(* IEC 61131-3 sources: AcpTrakStarwheel/Starlib, 9 files *)

(* ---- Types.typ ---- *)
TYPE
	FindClosestPcketSynReturnType : 	STRUCT
		ClosestPocket : UINT;
		NextClosestPocket : UINT;
	END_STRUCT;
END_TYPE

(*Star Target Calculations*)

TYPE
	slStarCalcTargetParType : 	STRUCT  (*Pocket sync position calculation parameters*)
		StarwheelRadius : REAL; (*Radius of the starwheel in mm*)
		StarwheelPeriod : REAL; (*Period of the starwheel in degrees*)
		StarwheelPocketCount : USINT; (*Number of pockets on the starwheel*)
		SectorTangentPos : REAL; (*Tangent position of the starwheel on the Trak sector*)
		DeltaT : TIME; (*Delay time to compensate in ms*)
	END_STRUCT;
	slStarCalcTargetInternalType : 	STRUCT  (*Internal Data*)
		TargetIndex : USINT; (*Index to generate a position for*)
		PeriodCount : INT; (*Number of periods being monitored*)
		CurrentStarwheelPeriod : INT; (*The current period of the target*)
		MultiturnPosition : REAL; (*The current multiturn position of the starwheel*)
		StarPosPredict : REAL; (*Starwheel predicted position*)
		OldStarPosPredict : REAL; (*Previously recorded predicted starwheel position*)
		AngleOffset : REAL; (*Angle offset of the starwheel compensating for pocket and period*)
		PocketAngle : REAL; (*Angle of the monitored pocket*)
		TrakSyncPosRaw : REAL; (*Raw trak position not accounting for the tangent position*)
		PerformCalculation : BOOL; (*Perform calculation while true*)
		State : slStarCalcTargetStateEnum; (*State of execution*)
	END_STRUCT;
	slStarCalcTargetStateEnum :
		( (*State of execution*)
		slTARGET_CALC_STATE_IDLE, (*Idle state*)
		slTARGET_CALC_STATE_RUN, (*Run state*)
		slTARGET_CALC_STATE_ERROR (*Error state*)
		);
END_TYPE

(*Star Pocket Sync*)

TYPE
	slStarPocketSyncParType : 	STRUCT  (*Pocket Sync Parameters*)
		StarCalcTarget : slStarCalcTargetParType; (*Calculation parameters*)
		CycPos : slStarPocketCycPosParType; (*Cyclic position parameters*)
		ResizeStart : McAcpTrakShResizeParamType; (*Resize dimensions at start of synchronization*)
		ResizeEnd : McAcpTrakShResizeParamType; (*Resize dimensions at end of synchronization*)
		Release : slStarPocketSyncReleaseParType; (*Release Parameters*)
	END_STRUCT;
	slStarPocketCycPosParType : 	STRUCT  (*Cyclic Position parameters*)
		AdvancedParameters : McAdvMoveCycParType; (*Advanced parameters*)
		InterpolationMode : McIplModeEnum; (*Interpolation mode*)
	END_STRUCT;
	slStarPocketSyncReleaseParType : 	STRUCT  (*Release motion parameters*)
		Position : LREAL; (*Release position on trak*)
		ResizePosition : LREAL; (*Resize position on trak after release*)
		Velocity : REAL; (*Release Velocity*)
		Acceleration : REAL; (*Release Acceleration*)
		Deceleration : REAL; (*Release Deceleration*)
		Jerk : REAL; (*Release Jerk*)
		Direction : McDirectionEnum; (*Release Direction*)
		BufferMode : McBufferModeEnum; (*Release Buffer Mode*)
	END_STRUCT;
	slStarPocketSyncInternalType : 	STRUCT  (*Internal Data*)
		StarCalcTarget : slStarCalcTarget; (*Calculate the sync position*)
		CycPos : MC_BR_ElasticMoveCycPos_AcpTrak; (*Synchronize the shuttle ot the position*)
		ShReadInfo : MC_BR_ShReadInfo_AcpTrak; (*Read shuttle information for its position*)
		MoveVel : MC_BR_ElasticMoveVel_AcpTrak; (*Release the shuttle from synchronization*)
		Resize : MC_BR_ShResize_AcpTrak; (*Resize the shuttle at start*)
		State : slStarPocketSyncStateEnum; (*State of execution*)
	END_STRUCT;
	slStarPocketSyncStateEnum :
		( (*State of execution*)
		slPOCKET_SYN_STATE_IDLE, (*Idle state*)
		slPOCKET_SYN_STATE_WAIT_SYNC, (*Wait for sync*)
		slPOCKET_SYN_STATE_RESIZE_START, (*Resize shuttle for start of sync*)
		slPOCKET_SYN_STATE_SYNC, (*Perform synchronization*)
		slPOCKET_SYN_STATE_RELEASE, (*Release shuttle*)
		slPOCKET_SYN_STATE_WAIT_RESIZE, (*Wait for the shuttle to reach the position to resize*)
		slPOCKET_SYN_STATE_RESIZE_END, (*Resize shuttle for end of sync*)
		slPOCKET_SYN_STATE_DONE, (*Star wheel operation complete*)
		slPOCKET_SYN_STATE_RESET_FB, (*Reset function blocks*)
		slPOCKET_SYN_STATE_WAIT_NOT_BUSY, (*Wait for function blocks to report not busy*)
		slPOCKET_SYN_STATE_ERROR (*Error state*)
		);
END_TYPE

(*Star Recovery*)

TYPE
	slStarRecoveryParType : 	STRUCT  (*Star recovery parameters*)
		ResizeStart : McAcpTrakShResizeParamType; (*Resize dimensions at start of synchronization*)
		ResizeEnd : McAcpTrakShResizeParamType; (*Resize dimensions at end of synchronization*)
		SyncFurtherInEnabled : BOOL;
		Release : slStarRecoveryParReleaseType; (*Recovery Release Parameters*)
		ProcessPointStartPosition : LREAL; (*Position on the sector of the process point that starts the synchronization*)
		StartOffset : LREAL; (*Offset from the process point before synchronizing*)
		PocketErrorTolerance : LREAL; (*Allowed pocket error tolerance*)
		UserData : slStarRecoveryParUserDataType; (*UserData parameters*)
		Backup : slStarRecoveryParBackupType;
		ShExtentToFront : LREAL;
		SectorTangentPos : REAL;
		MeshZoneStartPos : LREAL; (*Starwheel dimensions*)
		MeshZoneEndPos : LREAL;
	END_STRUCT;
	slStarRecoveryParBackupType : 	STRUCT  (*Recovery Release Parameters*)
		BackupTolerance : LREAL;
		ProcessPointStart : McProcessPointType; (*Position on the sector of the process point that starts the synchronization*)
		MoveToBarAcceleration : REAL;
		MoveToBarDeceleration : REAL;
		MoveToBarVelocity : REAL;
	END_STRUCT;
	slStarRecoveryParUserDataType : 	STRUCT  (*UserData parameters*)
		UserDataAddress : UDINT; (*Pointer to the user data buffer*)
		UserDataSize : UDINT; (*Size of the user data buffer*)
		SrcUserDataWriteAddress : UDINT; (*Source of the data to write to the user data buffer*)
		DstUserDataWriteAddress : UDINT; (*Destination within the user data buffer to write*)
		UserDataWriteSize : UDINT; (*Size of the data to write to the user data buffer*)
	END_STRUCT;
	slStarRecoveryParReleaseType : 	STRUCT  (*Recovery Release Parameters*)
		Position : LREAL; (*Release position of the starwheel*)
		Velocity : REAL; (*Recovery Velocity*)
		Acceleration : REAL; (*Recovery Acceleration*)
		Deceleration : REAL; (*Recovery Deceleration*)
		DestinationSector : McSectorType; (*Recovery Destination Sector*)
	END_STRUCT;
	slStarRecoveryInternalType : 	STRUCT  (*Internal Data*)
		Handle : UDINT; (*Handle to the starwheel internal data*)
		SecGetShuttle : MC_BR_SecGetShuttle_AcpTrak; (*Get shuttles on the sector*)
		ShResize : MC_BR_ShResize_AcpTrak; (*Resize shuttle*)
		RoutedMoveVel : MC_BR_RoutedMoveVel_AcpTrak; (*Send shuttle*)
		RoutedMoveAbs : MC_BR_RoutedMoveAbs_AcpTrak;
		ElasticMoveVel : MC_BR_ElasticMoveVel_AcpTrak; (*Send the shuttle*)
		ElasticMoveAbs : MC_BR_ElasticMoveAbs_AcpTrak;
		ShCopyUserData : MC_BR_ShCopyUserData_AcpTrak; (*Copy user data*)
		AsmGetInfo : MC_BR_AsmGetInfo_AcpTrak; (*Used to see if sectors are being simulated*)
		BarrierCmd : MC_BR_BarrierCommand_AcpTrak;
		OldRemainingCount : UINT; (*Previously recorded remaining count*)
		Data : slStarRecoveryInternalDataType; (*Data*)
		State : slStarRecoveryStateEnum; (*State of execution*)
		i : USINT; (*Index*)
	END_STRUCT;
	slStarRecoveryInternalDataFIType : 	STRUCT
		CurrentPocketIndex : UINT; (*Current pocket index being evaluated*)
	END_STRUCT;
	slStarRecoveryInternalDataType : 	STRUCT  (*Recovery data*)
		Init : slStarRecoverylDataInitType; (*Initial recovery data*)
		Mesh : slStarRecoveryDataMeshType;
		Sync : slStarRecoveryDataSyncType; (*Sync recovery data*)
		Backup : slStarRecoveryDataBackupType; (*Backup recovery data*)
		UserData : slStarRecoveryDataUserDataType;
		SyncFurtherIn : slStarRecoveryInternalDataFIType;
		PocketWidth : LREAL; (*Width of a pocket on the starwheel*)
	END_STRUCT;
	slStarRecoveryDataSyncFurInType : 	STRUCT
		LastSyncedPocket : USINT; (*Next open pocket available to sync further in*)
		LastSyncedPocketValid : BOOL;
	END_STRUCT;
	slStarRecoveryDataUserDataType : 	STRUCT
		UserDataWriteCount : UINT;
	END_STRUCT;
	slStarRecoverylDataInitType : 	STRUCT  (*Intial recovery data*)
		ShuttlePos : ARRAY[0..slMAX_SH_IDX_IN_SEC]OF LREAL; (*Shuttle positions found at initialization*)
		ShuttleAxis : ARRAY[0..slMAX_SH_IDX_IN_SEC]OF McAxisType; (*Shuttle axes found at initialization*)
		NumShuttles : UINT; (*Number of shuttles found at initialization*)
		ShuttleEvalCount : USINT; (*Number of shuttles found at initialization that have been evalueated*)
	END_STRUCT;
	slStarRecoveryDataMeshType : 	STRUCT  (*Sync recovery data*)
		PocketEvalIndex : UINT; (*Pocket index to evaluate*)
		PocketEvalIndexValid : BOOL;
		NextClosestPocketIndex : UINT;
		ClosestPocketTaken : BOOL;
		NextClosestPocketTaken : BOOL;
		PocketEvalCount : USINT; (*Number of pockets evaluated*)
		Axes : ARRAY[0..slMAX_SH_IDX_IN_SEC]OF McAxisType; (*Sync axes*)
		ShuttleErrors : ARRAY[0..slMAX_SH_IDX_IN_SEC]OF LREAL;
		PocketIndices : ARRAY[0..slMAX_SH_IDX_IN_SEC]OF UINT; (*Pocket indices assigned to the sync axes*)
		ShuttleError : LREAL; (*Distance from shuttle to pocket*)
		ShuttleErrorNew : LREAL; (*New distance from shuttle to pocket*)
		NextClosestPocketError : LREAL;
		RecoveredCount : UINT; (*Number of shuttles recovered*)
	END_STRUCT;
	slStarRecoveryDataSyncType : 	STRUCT  (*Sync recovery data*)
		PocketEvalIndex : UINT; (*Pocket index to evaluate*)
		PocketEvalIndexValid : BOOL;
		NextClosestPocketIndex : UINT;
		ClosestPocketTaken : BOOL;
		NextClosestPocketTaken : BOOL;
		PocketEvalCount : USINT; (*Number of pockets evaluated*)
		Axes : ARRAY[0..slMAX_SH_IDX_IN_SEC]OF McAxisType; (*Sync axes*)
		ShuttleErrors : ARRAY[0..slMAX_SH_IDX_IN_SEC]OF LREAL;
		PocketIndices : ARRAY[0..slMAX_SH_IDX_IN_SEC]OF UINT; (*Pocket indices assigned to the sync axes*)
		ShuttleError : LREAL; (*Distance from shuttle to pocket*)
		ShuttleErrorNew : LREAL; (*New distance from shuttle to pocket*)
		RecoveredCount : UINT; (*Number of shuttles recovered*)
		ShuttlePos : ARRAY[0..slMAX_SH_IDX_IN_SEC]OF LREAL; (*Shuttle positions found at initialization*)
		SyncFurtherIn : slStarRecoveryDataSyncFIType;
		NextClosestPocketError : LREAL;
	END_STRUCT;
	slStarRecoveryDataSyncFIType : 	STRUCT
		ClosestPocketToMeshFound : BOOL;
		ClosestPocketToMesh : UINT;
		NoClosestPocketFound : BOOL;
		FirstPocketInMeshIndex : UINT;
		FirstShuttleInMeshError : LREAL;
		FirstSyncPocketError : LREAL;
	END_STRUCT;
	slStarRecoveryDataBackupType : 	STRUCT  (*Backup recovery data*)
		EvalCount : USINT; (*Number of shuttles evaluated*)
		Axes : ARRAY[0..slMAX_SH_IDX_IN_SEC]OF McAxisType; (*Axes found in the backup area*)
		Positions : ARRAY[0..slMAX_SH_IDX_IN_SEC]OF LREAL;
		RecoveredCount : USINT; (*Number of shuttles recovered*)
		IsBeforeBarrier : ARRAY[0..slMAX_SH_IDX_IN_SEC]OF BOOL; (*Indicates if a shuttle is in the backup zone but before the barrier (have to move to gaurantee it won't get stuck at the barrier)*)
		MovedToBarrier : ARRAY[0..slMAX_SH_IDX_IN_SEC]OF BOOL; (*Indicated if a shuttle has been moved to the barrier location*)
		SyncFurtherIn : slStarRecoveryDataBackupFIType;
		Position : LREAL;
		PocketOvertakeIndex : UINT;
	END_STRUCT;
	slStarRecoveryDataBackupFIType : 	STRUCT  (*Sync further in type for backup zone*)
		CurrentPocketIndex : UINT; (*Current pocket index being evaluated*)
		SyncFurtherInFinished : BOOL; (*All shuttles in backup zone have synced to the closest pockets possible*)
	END_STRUCT;
	slStarRecoveryStateEnum :
		( (*State of execution*)
		slREC_STATE_IDLE, (*Idle state*)
		slREC_STATE_CHECK_SECTOR_SIM,
		slREC_STATE_GET_SHUTTLES, (*Get shuttles on the sector*)
		slREC_STATE_ATTACH_TO_SECTOR,
		slREC_STATE_GET_SHUTTLES_NEXT, (*Get the next shuttle on the sector*)
		slREC_STATE_RELEASE_ZONE_CHECK, (*Check for shuttles in the release zone*)
		slREC_STATE_RELEASE_ZONE_RESIZE, (*Resize shuttles in the release zone*)
		slREC_STATE_RELEASE_ZONE_SEND, (*Send shuttles in the release zone*)
		slREC_STATE_RELEASE_ZONE_NEXT, (*Get the next shuttle in the release zone*)
		slREC_STATE_MESH_ZONE_CHECK, (*Check for shuttles in the sync zone*)
		slREC_STATE_MESH_ZONE_TARGET, (*Assign target for sync*)
		slREC_STATE_MESH_ZONE_RESIZE, (*Resize shuttles*)
		slREC_STATE_MESH_ZONE_NEXT, (*Get the next shuttle in the sync zone*)
		slREC_STATE_SYN_ZONE_CHECK, (*Check for shuttles in the sync zone*)
		slREC_STATE_SYN_ZONE_TARGET, (*Assign target for sync*)
		slREC_STATE_SYN_ZONE_RESIZE, (*Resize shuttles*)
		slREC_STATE_SYN_ZONE_NEXT, (*Get the next shuttle in the sync zone*)
		slREC_STATE_BACKUP_ZONE_CHECK, (*Check for shuttles in the backup zone*)
		slREC_STATE_PBACKUP_ZONE_RSIZE, (*Resize shuttles in the backup zone*)
		slREC_STATE_PBACKUP_ZONE_SEND, (*Send shuttles in the backup zone*)
		slREC_STATE_PBACKUP_ZONE_NEXT, (*Get the next shuttle in the backup zone*)
		slREC_STATE_PBCKUP_ZNE_USR_DATAG, (*Get the next shuttle in the backup zone*)
		slREC_STATE_SYN_ZONE_SYNC, (*Sync shuttles in the sync zone*)
		slREC_STATE_MESH_ZONE_SYNC, (*Sync shuttles in the sync zone*)
		slREC_STATE_SYN_GET_USERDATA, (*Get sync zone userdata*)
		slREC_STATE_SYN_SET_USERDATA, (*Set sync zone userdata*)
		slREC_STATE_BACKUP_ZONE_TARGET, (*Wait for a target for shuttle in backup zone*)
		slREC_STATE_BACKUP_ZONE_BAROPEN, (*Wait for a target for shuttle in backup zone*)
		slREC_STATE_BACKUP_ZONE_MOVBAR,
		slREC_STATE_BACKUP_ZONE_BARCLOSE,
		slREC_STATE_BACKUP_ZONE_SYNC, (*Sync shuttle in backup zone to target*)
		slREC_STATE_BACKUP_ZONE_SYNC_FI, (*Backup zone sync further in*)
		slREC_STATE_BACKUP_GET_USERDATA, (*Get backup zone userdata*)
		slREC_STATE_BACKUP_SET_USERDATA, (*Set backup zone userdata*)
		slREC_STATE_GET_USERDATA,
		slREC_STATE_SET_USERDATA,
		slREC_STATE_FI_WAIT_SHUTTLE, (*Wait for a new shuttle to come by*)
		slREC_STATE_DONE, (*Recovery is complete*)
		slREC_STATE_WAIT_NOT_BUSY, (*Wait for function blocks to report not busy*)
		slREC_STATE_ERROR (*Error state*)
		);
END_TYPE

(*Star Sync*)

TYPE
	slStarSyncParType : 	STRUCT  (*Pocket Queue Parameters*)
		Landing : slStarSyncLandingParType; (*Landing parameters*)
		Starting : slStarSyncStartingParType; (*Starting parameters*)
		Staging : slStarSyncStagingParType; (*Staging parameters*)
		StartOffset : LREAL; (*Offset from the staging position before synchronizing*)
		SyncPar : slStarPocketSyncParType; (*Synchronization parameters*)
		Recovery : slStarSyncRecoveryParType; (*Star parameters for recovery*)
		Skip : slStarSyncSkipParType; (*Skip parameters*)
		ShExtentToFront : LREAL;
	END_STRUCT;
	slStarSyncLandingParType : 	STRUCT  (*Landing parameters*)
		Position : LREAL; (*Target Position*)
		Velocity : REAL; (*Target Velocity*)
		Acceleration : REAL; (*Target Acceleration*)
		Deceleration : REAL; (*Target Deceleration*)
		AdvancedParameters : McAcpTrakAdvRouteParType; (*Advanced move parameters*)
	END_STRUCT;
	slStarSyncStartingParType : 	STRUCT  (*Starting parameters*)
		Position : LREAL; (*Target Position*)
		Velocity : REAL; (*Target Velocity*)
	END_STRUCT;
	slStarSyncStagingParType : 	STRUCT  (*Staging parameters*)
		Position : LREAL; (*Target Position*)
		Velocity : REAL; (*Target Velocity*)
		Acceleration : REAL; (*Target Acceleration*)
		Deceleration : REAL; (*Target Deceleration*)
	END_STRUCT;
	slStarSyncRecoveryParType : 	STRUCT  (*Star parameters for recovery*)
		Release : slStarSyncRecoveryReleaseType; (*Release parameters*)
		UserData : slStarRecoveryParUserDataType; (*User data buffer data for successful recovery*)
		SyncFurtherInEnabled : BOOL;
		PocketErrorTolerance : LREAL; (*Pocket error tolerance for resynchronization*)
		MoveToBarVelocity : REAL;
		MoveToBarAcceleration : REAL;
		MoveToBarDeceleration : REAL;
		BackupTolerance : LREAL;
	END_STRUCT;
	slStarSyncRecoveryReleaseType : 	STRUCT  (*Release parameters*)
		Velocity : REAL; (*Recovery Velocity*)
		Acceleration : REAL; (*Recovery Acceleration*)
		Deceleration : REAL; (*Recovery Deceleration*)
		DestinationSector : McSectorType; (*Recovery Destination Sector*)
	END_STRUCT;
	slStarSyncSkipParType : 	STRUCT  (*Skip parameters*)
		NumSkips : USINT; (*Number of skips if skipping is enabled*)
		NumDisabled : USINT; (*Number of disabled pockets*)
		DisabledIdx : ARRAY[0..slMAX_DISABLE_POCKET_IDX]OF USINT; (*Disabled pockets*)
	END_STRUCT;
	slStarSyncCalcDataType : 	STRUCT
		StarPosPredict : REAL; (*Current starwheel position + predictive compensation*)
		CurrentStarwheelPeriod : INT; (*Current period of the 'real' starwheel, used to calculate a multiturn position*)
		MultiturnPosition : REAL; (*Current position of the 'virtual' starwheel*)
	END_STRUCT;
	slStarSyncInternalType : 	STRUCT  (*Internal Data*)
		TypeID : UDINT; (*Internal data type ID*)
		ErrorID : DINT; (*Last recorded error ID*)
		Recovery : slStarRecovery; (*Recovery process*)
		RecoveryPar : slStarRecoveryParType; (*Recovery parameters*)
		MaxTargetIndex : USINT; (*Highest pocket sync target index used*)
		LandingBuffer : tbAsyncShuttleBufferType; (*Buffer of shuttles that are landing on the sector*)
		StagingBuffer : tbAsyncShuttleBufferType; (*Buffer of shuttles that are being staged*)
		LandingBufferMan : tbRoutedMoveVelTrgBuffer; (*Landing shuttle buffer manager*)
		LandingBufferPar : tbRtdMvVelTrgBufferParType; (*Landing buffer parameters*)
		StagingBufferMan : tbElasticMoveAbsPosBuffer; (*Staging shuttle buffer manager*)
		StagingBufferPar : tbElaMvAbsPosBufferParType; (*Staging buffer parameters*)
		PocketSync : ARRAY[0..slMAX_TARGET_IDX]OF slStarPocketSync; (*Pocket Sync Targets*)
		LastPocketActiveState : ARRAY[0..slMAX_TARGET_IDX]OF BOOL; (*Capture the last pocket sync active state*)
		LastTargetPosition : ARRAY[0..slMAX_TARGET_IDX]OF REAL; (*Last observed target position for each target*)
		NextSyncTarget : UINT; (*Next target to sync shuttle with*)
		NewDisabledOvertake : BOOL; (*A disabled target position has passed the synchronization threshold*)
		NewOvertakeDetected : BOOL; (*A target position has passed the synchronization threshold*)
		State : slStarSyncStateEnum; (*State of execution*)
		SkipCount : USINT; (*Number of pockets skipped*)
		PocketDisabled : BOOL; (*Current target pocket is disabled*)
		PeriodCount : USINT; (*Number of periods to monitor*)
		i : UINT; (*Index*)
		n : USINT; (*Index*)
		PocketSyncBusy : BOOL; (*Temporary variable to determine if a pocket sync is still busy*)
		PocketSyncError : BOOL; (*Temporary variable to determine if a pocket sync has an error*)
		PocketSyncErrorID : DINT; (*Temporary variable to determine the pocket sync error ID*)
		NextSyncFITarget : UINT; (*Next sync further in target found*)
		SyncFurtherInDone : BOOL;
		MeshZoneStartPos : LREAL;
		MeshZoneEndPos : LREAL;
		PocketWidth : LREAL;
		RecoveryDone : BOOL;
		StarCalcData : slStarSyncCalcDataType; (*Includes Calc Target information that is Starwheel-specific, rather than Pocket-specific*)
		OldStarPosPredict : REAL; (*Star Position, including predictive compensation, from last cycle*)
		Status : DINT; (*Status*)
	END_STRUCT;
	slStarSyncStateEnum :
		( (*State of execution*)
		slSTAR_STATE_INIT, (*Initialize handle and data*)
		slSTAR_STATE_IDLE, (*Idle state*)
		slSTAR_STATE_RECOVER, (*Recover shuttles*)
		slSTAR_STATE_WAIT_TARGET, (*Wait for the next target to arrive*)
		slSTAR_STATE_WAIT_SHUTTLE, (*Wait for the next shuttle to arrive*)
		slSTAR_STATE_SYNC, (*Sync shuttle to pocket*)
		slSTAR_STATE_RESET_FB, (*Reset function blocks*)
		slSTAR_STATE_WAIT_NOT_BUSY, (*Wait for function blocks to report not busy*)
		slSTAR_STATE_ERROR (*An error occurred*)
		);
END_TYPE

(*Get Shuttle*)

TYPE
	slStarGetShuttleInternalType : 	STRUCT  (*Internal Data*)
		i : USINT; (*Index*)
		Present : BOOL; (*Temporary shuttle presence*)
		Axis : McAxisType; (*Temporary Axis Handle*)
		Position : REAL; (*Temporary Position*)
	END_STRUCT;
END_TYPE

(*Star Sync Diagnostics*)

TYPE
	slStarDiagType : 	STRUCT  (*Output starwheel diagnostics*)
		AngleOffset : ARRAY[0..slMAX_TARGET_IDX]OF REAL; (*Angle offsets of synchronization targets*)
		PocketAngle : ARRAY[0..slMAX_TARGET_IDX]OF REAL; (*Pocket angles of synchronization targets*)
		TrackSyncRaw : ARRAY[0..slMAX_TARGET_IDX]OF REAL; (*Raw synchronization positions of synchronization targets*)
		TrackSyncLast : ARRAY[0..slMAX_TARGET_IDX]OF REAL; (*Last synchronization positions of synchronization targets*)
		TrackSyncPos : ARRAY[0..slMAX_TARGET_IDX]OF REAL; (*Current synchronization positions of synchronization targets*)
		TargetAssigned : ARRAY[0..slMAX_TARGET_IDX]OF BOOL; (*A shuttle has been assigned to the synchronization target*)
		TargetInSync : ARRAY[0..slMAX_TARGET_IDX]OF BOOL; (*A shuttle is in sync with the synchronization target*)
		TargetInSyncLast : ARRAY[0..slMAX_TARGET_IDX]OF BOOL; (*Last In Sync status of synchronization target*)
	END_STRUCT;
	slStarDiagInternalType : 	STRUCT  (*Internal Data*)
		Handle : UDINT; (*Starwheel handle*)
		i : UINT; (*Index*)
		State : slStarDiagStateEnum; (*State of execution*)
	END_STRUCT;
	slStarDiagStateEnum :
		( (*State of execution*)
		slSTAR_DIAG_STATE_IDLE, (*Idle state*)
		slSTAR_DIAG_STATE_RUNNING, (*Running state*)
		slSTAR_DIAG_STATE_ERROR (*Error state*)
		);
END_TYPE

(*Star Sync Diagnostics Last State Error*)

TYPE
	slStarDiagLastStateInternalType : 	STRUCT  (*Internal data*)
		LastStateData : slStarDiagStateType; (*Last recorded state data*)
		State : slStarDiagStateEnum; (*State of execution*)
		Handle : UDINT; (*Starwheel handle*)
		i : UINT; (*Index*)
		StarRecoveryError : BOOL; (*Last star recovery error status*)
		StarPocketSyncError : ARRAY[0..slMAX_TARGET_IDX]OF BOOL; (*Last star pocket sync error status*)
		StarCalcTargetError : ARRAY[0..slMAX_TARGET_IDX]OF BOOL; (*Last calc target error status*)
	END_STRUCT;
	slStarDiagStateType : 	STRUCT  (*States of the star function blocks*)
		StarSync : slStarSyncStateEnum; (*Star state*)
		StarSyncAtReset : slStarSyncStateEnum; (*Star state before entering reset state*)
		StarRecovery : slStarRecoveryStateEnum; (*Recovery state*)
		StarPocketSync : ARRAY[0..slMAX_TARGET_IDX]OF slStarPocketSyncStateEnum; (*Star Pocket state*)
		StarCalcTarget : ARRAY[0..slMAX_TARGET_IDX]OF slStarCalcTargetStateEnum; (*Calc target state*)
	END_STRUCT;
	slStarDiagErrorIDType : 	STRUCT  (*Error IDs at last error*)
		StarSync : DINT; (*Recorded sync error*)
		StarRecovery : DINT; (*Recorded recovery error*)
		StarPocketSync : ARRAY[0..slMAX_TARGET_IDX]OF DINT; (*Recorded pocket sync error*)
		StarCalcTarget : ARRAY[0..slMAX_TARGET_IDX]OF DINT; (*Recorded calc target error*)
	END_STRUCT;
END_TYPE

(*Star Sync Diagnostices State Trace*)

TYPE
	slStarDiagStateTraceStatesType : 	STRUCT  (*State data*)
		StarSync : slStarDiagStateTraceStarSyncType; (*Star Sync State trace data*)
		StarRecovery : slStarDiagStateTraceStarRecType; (*Star Recovery State trace data*)
		StarPocket : ARRAY[0..slMAX_TARGET_IDX]OF slStarDiagStateTraceStarPockType; (*Star Pocket State trace data*)
		StarCalc : ARRAY[0..slMAX_TARGET_IDX]OF slStarDiagStateTraceStarCalcType;
	END_STRUCT;
	slStarDiagStateTraceStarSyncType : 	STRUCT  (*Star Sync State trace data*)
		LastIndex : USINT; (*Last index with a valid state*)
		State : ARRAY[0..slMAX_STATE_TRACE_IDX]OF slStarSyncStateEnum; (*Star Sync trace data*)
	END_STRUCT;
	slStarDiagStateTraceStarRecType : 	STRUCT  (*Star Recovery State trace data*)
		LastIndex : USINT; (*Last index with a valid state*)
		State : ARRAY[0..slMAX_STATE_TRACE_IDX]OF slStarRecoveryStateEnum; (*Star Recovery trace data*)
	END_STRUCT;
	slStarDiagStateTraceStarPockType : 	STRUCT  (*Star Pocket State trace data*)
		LastIndex : USINT; (*Last index with a valid state*)
		State : ARRAY[0..slMAX_STATE_TRACE_IDX]OF slStarPocketSyncStateEnum; (*Star Pocket trace data*)
	END_STRUCT;
	slStarDiagStateTraceStarCalcType : 	STRUCT  (*Star Calc State trace data*)
		LastIndex : USINT; (*Last index with a valid state*)
		State : ARRAY[0..slMAX_STATE_TRACE_IDX]OF slStarCalcTargetStateEnum; (*Star Calc trace data*)
	END_STRUCT;
	slStarDiagStateTraceInternalType : 	STRUCT  (*Internal Data*)
		Handle : UDINT; (*Starwheel handle*)
		i : UINT; (*Index*)
		State : slStarDiagStateEnum; (*State of execution*)
	END_STRUCT;
END_TYPE

(* ---- ClosestSyncPocket.st ---- *)
(* Finds the closest pocket to the start of the mesh zone of the starwheel that a shuttle can sync to *)
FUNCTION ClosestSyncPocket

    StarInternal ACCESS Handle;

    FOR i := 0 TO StarInternal.MaxTargetIndex DO
        TangentPocketLocationErrorNew := StarInternal.PocketSync[i].TargetPosition - MeshZoneStartPos;
        FirstSyncPocketLocationErrorNew := StarInternal.PocketSync[i].TargetPosition - SyncZoneStartPos;
        IF i = 0 THEN
            TangentPocketLocationError := TangentPocketLocationErrorNew;
            FirstSyncPocketLocationError    := FirstSyncPocketLocationErrorNew;
        END_IF;

        IF ABS(TangentPocketLocationErrorNew) < ABS(TangentPocketLocationError) AND (StarInternal.PocketSync[i].TargetPosition <= MeshZoneStartPos) THEN
            TangentPocketIndex := i;
            TangentPocketLocationError := TangentPocketLocationErrorNew;
        END_IF

        IF ABS(FirstSyncPocketLocationErrorNew) < ABS(FirstSyncPocketLocationError) AND StarInternal.PocketSync[i].TargetPosition >= SyncZoneStartPos THEN
            FirstSyncPocketIndex := i;
            FirstSyncPocketLocationError := FirstSyncPocketLocationErrorNew;
        END_IF
    END_FOR

    CurrentEvalPocket   := FirstSyncPocketIndex;
    PrevEvalPocket      := FirstSyncPocketIndex;
    FOR i := 0 TO StarInternal.MaxTargetIndex DO
        IF (CurrentEvalPocket = TangentPocketIndex) OR (StarInternal.PocketSync[CurrentEvalPocket].Sync) THEN
            CurrentEvalPocket   := PrevEvalPocket;
            EXIT;
        ELSE
            CurrentEvalPocketValid  := TRUE;
            ClosestSyncPocket   := CurrentEvalPocket;
        END_IF;

        PrevEvalPocket  := CurrentEvalPocket;
        IF CurrentEvalPocket = 0 THEN
            CurrentEvalPocket   := StarInternal.MaxTargetIndex;
        ELSE
            CurrentEvalPocket   := CurrentEvalPocket - 1;
        END_IF;
    END_FOR;

    IF NOT CurrentEvalPocketValid THEN
        ClosestSyncPocket   := slNO_CLOSEST_POCKET_FOUND;
    END_IF;

END_FUNCTION

(* ---- StarDiagLastStateError.st ---- *)
FUNCTION_BLOCK slStarDiagLastStateError

    CASE Internal.State OF

        slSTAR_DIAG_STATE_IDLE:

            IF Enable THEN
                Busy := 1;
                IF Handle = 0 THEN
                    Error := 1;
                    ErrorID := slERR_INVALID_HANDLE;
                    Internal.State := slSTAR_DIAG_STATE_ERROR;
                ELSE
                    Internal.Handle := Handle;
                    StarInternal ACCESS Internal.Handle;
                    IF StarInternal.TypeID <> slSTAR_INTERNAL_TYPE_ID THEN
                        Error := 1;
                        ErrorID := slERR_INVALID_HANDLE;
                        Internal.State := slSTAR_DIAG_STATE_ERROR;
                    ELSE
                        brsmemset(ADR(ErrorIDs), 0, SIZEOF(ErrorIDs));
                        Internal.LastStateData.StarSync := StarInternal.State;
                        Internal.LastStateData.StarRecovery := StarInternal.Recovery.Internal.State;
                        LastStates.StarSync := slSTAR_STATE_IDLE;
                        LastStates.StarRecovery := slREC_STATE_IDLE;
                        FOR Internal.i := 0 TO slMAX_TARGET_IDX DO
                            Internal.LastStateData.StarPocketSync[Internal.i] := StarInternal.PocketSync[Internal.i].Internal.State;
                            Internal.LastStateData.StarCalcTarget[Internal.i] := StarInternal.PocketSync[Internal.i].Internal.StarCalcTarget.Internal.State;
                            LastStates.StarPocketSync[Internal.i] := slPOCKET_SYN_STATE_IDLE;
                            LastStates.StarCalcTarget[Internal.i] := slTARGET_CALC_STATE_IDLE;
                        END_FOR
                        Internal.State := slSTAR_DIAG_STATE_RUNNING;
                    END_IF
                END_IF
            END_IF

        slSTAR_DIAG_STATE_RUNNING:

            IF Enable THEN
                StarInternal ACCESS Internal.Handle;
                //Monitor the star sync state
                IF (StarInternal.State = slSTAR_STATE_RESET_FB) AND (Internal.LastStateData.StarSync <> slSTAR_STATE_RESET_FB) THEN
                    Internal.LastStateData.StarSyncAtReset := Internal.LastStateData.StarSync;
                END_IF
                IF (StarInternal.State = slSTAR_STATE_ERROR) AND (Internal.LastStateData.StarSync <> slSTAR_STATE_ERROR) THEN
                    LastStates.StarSync := Internal.LastStateData.StarSyncAtReset;
                    ErrorIDs.StarSync := StarInternal.ErrorID;
                END_IF
                Internal.LastStateData.StarSync := StarInternal.State;
                //Monitor the star recovery state
                IF StarInternal.Recovery.Error AND NOT Internal.StarRecoveryError THEN
                    LastStates.StarRecovery := Internal.LastStateData.StarRecovery;
                    ErrorIDs.StarRecovery := StarInternal.Recovery.ErrorID;
                END_IF
                Internal.LastStateData.StarRecovery := StarInternal.Recovery.Internal.State;
                Internal.StarRecoveryError := StarInternal.Recovery.Error;
                FOR Internal.i := 0 TO slMAX_TARGET_IDX DO
                    //Monitor the pocket sync states
                    IF StarInternal.PocketSync[Internal.i].Error AND NOT Internal.StarPocketSyncError[Internal.i] THEN
                        LastStates.StarPocketSync[Internal.i] := Internal.LastStateData.StarPocketSync[Internal.i];
                        ErrorIDs.StarPocketSync[Internal.i] := StarInternal.PocketSync[Internal.i].ErrorID;
                    END_IF
                    Internal.LastStateData.StarPocketSync[Internal.i] := StarInternal.PocketSync[Internal.i].Internal.State;
                    Internal.StarPocketSyncError[Internal.i] := StarInternal.PocketSync[Internal.i].Error;
                    //Monitor the target calculation states
                    IF StarInternal.PocketSync[Internal.i].Internal.StarCalcTarget.Error AND NOT Internal.StarCalcTargetError[Internal.i] THEN
                        LastStates.StarCalcTarget[Internal.i] := Internal.LastStateData.StarCalcTarget[Internal.i];
                        ErrorIDs.StarCalcTarget[Internal.i] := StarInternal.PocketSync[Internal.i].Internal.StarCalcTarget.ErrorID;
                    END_IF
                    Internal.LastStateData.StarCalcTarget[Internal.i] := StarInternal.PocketSync[Internal.i].Internal.StarCalcTarget.Internal.State;
                    Internal.StarCalcTargetError[Internal.i] := StarInternal.PocketSync[Internal.i].Internal.StarCalcTarget.Error;
                END_FOR
                Valid := 1;
            ELSE
                Internal.StarRecoveryError := 0;
                brsmemset(ADR(Internal.StarPocketSyncError), 0, SIZEOF(Internal.StarPocketSyncError));
                brsmemset(ADR(Internal.StarCalcTargetError), 0, SIZEOF(Internal.StarCalcTargetError));
                Valid := 0;
                Busy := 0;
                Internal.State := slSTAR_DIAG_STATE_IDLE;
            END_IF

        slSTAR_DIAG_STATE_ERROR:

            IF NOT Enable THEN
                Error := 0;
                ErrorID := ERR_OK;
                Internal.State := slSTAR_DIAG_STATE_IDLE;
                Busy := 0;
            END_IF

    END_CASE

END_FUNCTION_BLOCK

(* ---- StarDiagStateTrace.st ---- *)
FUNCTION_BLOCK slStarDiagStateTrace

    CASE Internal.State OF

        slSTAR_DIAG_STATE_IDLE:

            IF Enable THEN
                Busy := 1;
                IF Handle = 0 THEN
                    Error := 1;
                    ErrorID := slERR_INVALID_HANDLE;
                    Internal.State := slSTAR_DIAG_STATE_ERROR;
                ELSE
                    Internal.Handle := Handle;
                    StarInternal ACCESS Internal.Handle;
                    IF StarInternal.TypeID <> slSTAR_INTERNAL_TYPE_ID THEN
                        Error := 1;
                        ErrorID := slERR_INVALID_HANDLE;
                        Internal.State := slSTAR_DIAG_STATE_ERROR;
                    ELSE
                        brsmemset(ADR(StateData), 0, SIZEOF(StateData));
                        StateData.StarSync.State[0] := StarInternal.State;
                        StateData.StarRecovery.State[0] := StarInternal.Recovery.Internal.State;
                        FOR Internal.i := 0 TO slMAX_TARGET_IDX DO
                            StateData.StarPocket[Internal.i].State[0] := StarInternal.PocketSync[Internal.i].Internal.State;
                            StateData.StarCalc[Internal.i].State[0] := StarInternal.PocketSync[Internal.i].Internal.StarCalcTarget.Internal.State;
                        END_FOR
                        Valid := 1;
                        Internal.State := slSTAR_DIAG_STATE_RUNNING;
                    END_IF
                END_IF
            END_IF

        slSTAR_DIAG_STATE_RUNNING:

            StarInternal ACCESS Internal.Handle;

            IF Enable THEN
                //Get the star sync state
                IF StarInternal.State <> StateData.StarSync.State[StateData.StarSync.LastIndex] THEN
                    StateData.StarSync.LastIndex := StateData.StarSync.LastIndex + 1;
                    IF StateData.StarSync.LastIndex > slMAX_STATE_TRACE_IDX THEN
                        StateData.StarSync.LastIndex := 0;
                    END_IF
                    StateData.StarSync.State[StateData.StarSync.LastIndex] := StarInternal.State;
                END_IF
                //Get the star recovery state
                IF StarInternal.Recovery.Internal.State <> StateData.StarRecovery.State[StateData.StarRecovery.LastIndex] THEN
                    StateData.StarRecovery.LastIndex := StateData.StarRecovery.LastIndex + 1;
                    IF StateData.StarRecovery.LastIndex > slMAX_STATE_TRACE_IDX THEN
                        StateData.StarRecovery.LastIndex := 0;
                    END_IF
                    StateData.StarRecovery.State[StateData.StarRecovery.LastIndex] := StarInternal.Recovery.Internal.State;
                END_IF
                FOR Internal.i := 0 TO slMAX_TARGET_IDX DO
                    //Get the pocket state
                    IF StarInternal.PocketSync[Internal.i].Internal.State <> StateData.StarPocket[Internal.i].State[StateData.StarPocket[Internal.i].LastIndex] THEN
                        StateData.StarPocket[Internal.i].LastIndex := StateData.StarPocket[Internal.i].LastIndex + 1;
                        IF StateData.StarPocket[Internal.i].LastIndex > slMAX_STATE_TRACE_IDX THEN
                            StateData.StarPocket[Internal.i].LastIndex := 0;
                        END_IF
                        StateData.StarPocket[Internal.i].State[StateData.StarPocket[Internal.i].LastIndex] := StarInternal.PocketSync[Internal.i].Internal.State;
                    END_IF
                    //Get the calc state
                    IF StarInternal.PocketSync[Internal.i].Internal.StarCalcTarget.Internal.State <> StateData.StarCalc[Internal.i].State[StateData.StarCalc[Internal.i].LastIndex] THEN
                        StateData.StarCalc[Internal.i].LastIndex := StateData.StarCalc[Internal.i].LastIndex + 1;
                        IF StateData.StarCalc[Internal.i].LastIndex > slMAX_STATE_TRACE_IDX THEN
                            StateData.StarCalc[Internal.i].LastIndex := 0;
                        END_IF
                       StateData.StarCalc[Internal.i].State[StateData.StarCalc[Internal.i].LastIndex] := StarInternal.PocketSync[Internal.i].Internal.StarCalcTarget.Internal.State;
                    END_IF
                END_FOR
            ELSE
                Valid := 0;
                Busy := 0;
                Internal.State := slSTAR_DIAG_STATE_IDLE;
            END_IF

        slSTAR_DIAG_STATE_ERROR:

            IF NOT Enable THEN
                Error := 0;
                ErrorID := ERR_OK;
                Internal.State := slSTAR_DIAG_STATE_IDLE;
                Busy := 0;
            END_IF

    END_CASE

END_FUNCTION_BLOCK

(* ---- StarLib.fun ---- *)
{REDUND_ERROR} FUNCTION EuclideanModuloFLT : REAL (*Implements Euclidean Modulo*)
	VAR_INPUT
		Dividend : REAL; (*Modulo Dividend*)
		Divisor : REAL; (*Modulo Divisor*)
	END_VAR
END_FUNCTION

{REDUND_ERROR} FUNCTION EuclideanModuloINT : INT (*Implements Euclidean Modulo*) (*$GROUP=User,$CAT=User,$GROUPICON=User.png,$CATICON=User.png*)
	VAR_INPUT
		Dividend : INT; (*Modulo Dividend*)
		Divisor : INT; (*Modulo Divisor*)
	END_VAR
END_FUNCTION

{REDUND_ERROR} FUNCTION ClosestSyncPocket : UINT (*Finds the closest pocket to the tangent point of the starwheel that a shuttle can sync to*) (*$GROUP=User,$CAT=User,$GROUPICON=User.png,$CATICON=User.png*)
	VAR_INPUT
		MeshZoneStartPos : LREAL; (*Tangent point of the starwheel*)
		SyncZoneStartPos : LREAL; (*Start of the sync zone on the starwheel sector*)
		Handle : UDINT; (*Starwheel internal data handle*)
	END_VAR
	VAR
		StarInternal : REFERENCE TO slStarSyncInternalType; (*Star Internal Data*)
		TangentPocketLocationError : LREAL; (*Error of the current evaluation pocket*)
		TangentPocketLocationErrorNew : LREAL;
		FirstSyncPocketLocationError : LREAL; (*Error of the current evaluation pocket*)
		FirstSyncPocketLocationErrorNew : LREAL;
		TangentPocketIndex : UINT;
		FirstSyncPocketIndex : UINT;
		CurrentEvalPocket : UINT;
		PrevEvalPocket : UINT;
		CurrentEvalPocketValid : BOOL;
		i : USINT;
	END_VAR
END_FUNCTION

{REDUND_ERROR} FUNCTION PocketOvertakeDetect : UINT (*Returns the pocket index of pocket that has crossed a point input to the function*) (*$GROUP=User,$CAT=User,$GROUPICON=User.png,$CATICON=User.png*)
	VAR_INPUT
		Handle : UDINT; (*Starwheel internal data handle*)
		Position : LREAL; (*Position that is being monitored for an overtake*)
	END_VAR
	VAR
		StarInternal : REFERENCE TO slStarSyncInternalType;
		i : UINT;
	END_VAR
END_FUNCTION

FUNCTION_BLOCK slStarCalcTarget (*Synchronous function block that calculates the position of the sync positions*)
	VAR_INPUT
		TargetIndex : USINT; (*Index to generate a position for*)
		PeriodCount : USINT; (*Number of periods to monitor*)
		Enable : BOOL; (*Calculate when true*)
		CalcData : REFERENCE TO slStarSyncCalcDataType;
		Parameters : REFERENCE TO slStarCalcTargetParType; (*Calculation parameters*)
	END_VAR
	VAR_OUTPUT
		Valid : BOOL; (*Position is valid*)
		TrakPos : REAL; (*Position on the trak*)
		Error : BOOL; (*An error occurred*)
		ErrorID : DINT; (*ID of the error that occurred*)
	END_VAR
	VAR
		Internal : slStarCalcTargetInternalType; (*Internal data*)
	END_VAR
END_FUNCTION_BLOCK

FUNCTION_BLOCK slStarPocketSync (*Synchronize a shuttle with a pocket*)
	VAR_INPUT
		TargetIndex : USINT; (*Index to generate a position for*)
		PeriodCount : USINT; (*Number of periods to monitor*)
		Enable : BOOL; (*Enable syncing to the pocket*)
		Axis : {REDUND_UNREPLICABLE} McAxisType; (*Shuttle to sync with pocket*)
		Sync : BOOL; (*Synchronize on rising edge*)
		CalcData : REFERENCE TO slStarSyncCalcDataType;
		Parameters : REFERENCE TO slStarPocketSyncParType; (*Pocket Sync Parameters*)
	END_VAR
	VAR_OUTPUT
		Busy : BOOL; (*Function Block is busy and must continue to be called*)
		Active : BOOL; (*The function block is active and ready for sync*)
		InSync : BOOL; (*The shuttle is in synchronization with the target position*)
		Done : BOOL; (*The shuttle is through the starwheel*)
		TargetPosition : REAL; (*The current target position*)
		Error : BOOL; (*An error occurred*)
		ErrorID : DINT; (*ID of the error that occurred*)
	END_VAR
	VAR
		Internal : slStarPocketSyncInternalType; (*Internal Data*)
	END_VAR
END_FUNCTION_BLOCK

FUNCTION_BLOCK slStarSync (*Star synchronization*)
	VAR_INPUT
		Sector : REFERENCE TO McSectorType; (*Sector for starwheel*)
		Assembly : REFERENCE TO McAssemblyType;
		ProcessPoint : REFERENCE TO McProcessPointType; (*Process point at the start of the sector*)
		Enable : BOOL; (*Enable starwheel*)
		SkipPockets : BOOL; (*Skip pockets when true*)
		DisablePockets : BOOL; (*Disable configured pockets when true*)
		StarwheelPosition : {REDUND_UNREPLICABLE} REAL; (*Position of the starwheel in degrees*)
		StarwheelVelocity : {REDUND_UNREPLICABLE} REAL; (*Velocity of the starwheel in degrees per second*)
		Parameters : REFERENCE TO slStarSyncParType; (*Queue parameters*)
	END_VAR
	VAR_OUTPUT
		Busy : BOOL; (*The function block is busy and must continue to be called*)
		ReadyForStart : BOOL; (*The function block is ready for starwheel movement*)
		Active : BOOL; (*Starwheel is active*)
		Handle : UDINT; (*Starwheel internal data handle*)
		Error : BOOL; (*An error occurred*)
		ErrorID : DINT; (*ID of the error that occurred*)
	END_VAR
	VAR
		Internal : slStarSyncInternalType; (*Internal Data*)
	END_VAR
END_FUNCTION_BLOCK

FUNCTION_BLOCK slStarRecovery (*Recover shuttles in the starwheel*)
	VAR_INPUT
		Sector : REFERENCE TO McSectorType; (*Sector for starwheel*)
		Assembly : REFERENCE TO McAssemblyType;
		Parameters : REFERENCE TO slStarRecoveryParType; (*Starwheel recovery parameters*)
		Handle : UDINT; (*Starwheel internal data handle*)
		Enable : BOOL; (*Enable recovery process*)
	END_VAR
	VAR_OUTPUT
		Busy : BOOL; (*The function block is busy and must continue to be called*)
		ReadyForStart : BOOL; (*The function block is ready for starwheel movement*)
		Done : BOOL; (*Recovery is complete*)
		Error : BOOL; (*An error occurred*)
		ErrorID : DINT; (*ID of the error that occurred*)
	END_VAR
	VAR
		Internal : slStarRecoveryInternalType; (*Internal Data*)
		StarInternal : REFERENCE TO slStarSyncInternalType; (*Star Internal Data*)
	END_VAR
END_FUNCTION_BLOCK

FUNCTION_BLOCK slStarGetShuttle (*Get the shuttle in a starwheel that is between two positions*)
	VAR_INPUT
		TrakPositionStart : REAL; (*Start position to look for the shuttle*)
		TrakPositionEnd : REAL; (*End position to look for the shuttle*)
		Handle : UDINT; (*Handle of the star sync to evaluate*)
		Enable : BOOL; (*Execute on a rising edge*)
	END_VAR
	VAR_OUTPUT
		Valid : BOOL; (*The shuttle and position are valid*)
		ShuttlePresent : BOOL; (*A shuttle is present between the two positions*)
		Axis : McAxisType; (*Shuttle Axis*)
		Position : REAL; (*Target position of the shuttle*)
		Error : BOOL; (*An error occurred*)
		ErrorID : DINT; (*ID of the error that occurred*)
	END_VAR
	VAR
		Internal : slStarGetShuttleInternalType; (*Internal Data*)
		StarInternal : REFERENCE TO slStarSyncInternalType; (*Star Internal Data*)
	END_VAR
END_FUNCTION_BLOCK

FUNCTION_BLOCK slStarDiag (*Star diagnostics*)
	VAR_INPUT
		Handle : UDINT; (*Starwheel handle*)
		Enable : BOOL; (*Enable outputting diagnostics*)
	END_VAR
	VAR_OUTPUT
		Busy : BOOL; (*The function block is busy and must continue to be called*)
		Valid : BOOL; (*The Diagnostic data is valid*)
		Diag : slStarDiagType; (*Diagnostic information*)
		Error : BOOL; (*An error occurred*)
		ErrorID : DINT; (*ID of the error that occurred*)
	END_VAR
	VAR
		Internal : slStarDiagInternalType; (*Internal Handle*)
		StarInternal : REFERENCE TO slStarSyncInternalType; (*Star Internal Data*)
	END_VAR
END_FUNCTION_BLOCK

FUNCTION_BLOCK slStarDiagLastStateError (*Get the last state before an error*)
	VAR_INPUT
		Handle : UDINT; (*Starwheel handle*)
		Enable : BOOL; (*Enable capturing the last state before an error*)
	END_VAR
	VAR_OUTPUT
		Busy : BOOL; (*The function block is busy and must continue to be called*)
		Valid : BOOL; (*The Diagnostic data is valid*)
		LastStates : slStarDiagStateType; (*Last states recorded before an error*)
		ErrorIDs : slStarDiagErrorIDType; (*Error IDs recorded on the last error*)
		Error : BOOL; (*An error occurred*)
		ErrorID : DINT; (*ID of the error that occurred*)
	END_VAR
	VAR
		Internal : slStarDiagLastStateInternalType; (*Internal Handle*)
		StarInternal : REFERENCE TO slStarSyncInternalType; (*Star Internal Data*)
	END_VAR
END_FUNCTION_BLOCK

FUNCTION_BLOCK slStarDiagStateTrace (*Trace the starwheel states*)
	VAR_INPUT
		Handle : UDINT; (*Starwheel handle*)
		Enable : BOOL; (*Enable capturing the last state before an error*)
	END_VAR
	VAR_OUTPUT
		Busy : BOOL; (*The function block is busy and must continue to be called*)
		Valid : BOOL; (*The State data is valid*)
		StateData : slStarDiagStateTraceStatesType; (*State trace*)
		Error : BOOL; (*An error occurred*)
		ErrorID : DINT; (*ID of the error that occurred*)
	END_VAR
	VAR
		Internal : slStarDiagStateTraceInternalType; (*Internal Handle*)
		StarInternal : REFERENCE TO slStarSyncInternalType; (*Star Internal Data*)
	END_VAR
END_FUNCTION_BLOCK

(* ---- StarPocketSync.st ---- *)
FUNCTION_BLOCK slStarPocketSync

    Internal.StarCalcTarget();

    TargetPosition := Internal.StarCalcTarget.TrakPos;

    CASE Internal.State OF

        slPOCKET_SYN_STATE_IDLE:

            IF Enable THEN

                Busy := 1;

                Internal.StarCalcTarget.TargetIndex := TargetIndex;
				Internal.StarCalcTarget.PeriodCount := PeriodCount;
				Internal.StarCalcTarget.CalcData := ADR(CalcData);
                Internal.StarCalcTarget.Parameters := ADR(Parameters.StarCalcTarget);
                Internal.StarCalcTarget.Enable := 1;

                Internal.State := slPOCKET_SYN_STATE_WAIT_SYNC;

            END_IF

        slPOCKET_SYN_STATE_WAIT_SYNC:

            IF NOT Enable THEN
                Internal.State := slPOCKET_SYN_STATE_RESET_FB;
            ELSIF Internal.StarCalcTarget.Error THEN
                Error := 1;
                ErrorID := Internal.StarCalcTarget.ErrorID;
                Internal.State := slPOCKET_SYN_STATE_RESET_FB;
            ELSIF Sync THEN

                Internal.CycPos.Axis := ADR(Axis);
                Internal.CycPos.AdvancedParameters := Parameters.CycPos.AdvancedParameters;
                Internal.CycPos.InterpolationMode := Parameters.CycPos.InterpolationMode;

                Internal.ShReadInfo.Axis := ADR(Axis);
                Internal.ShReadInfo.Enable := 1;

                Internal.Resize.Axis := ADR(Axis);
                Internal.Resize.Command := mcACPTRAK_RESIZE_DIMENSIONS;
                Internal.Resize.ResizeParameter := Parameters.ResizeStart;
                Internal.Resize.Execute := 1;

                Internal.MoveVel.Axis := ADR(Axis);
                Internal.MoveVel.Velocity := Parameters.Release.Velocity;
                Internal.MoveVel.Acceleration := Parameters.Release.Acceleration;
                Internal.MoveVel.Deceleration := Parameters.Release.Deceleration;
                Internal.MoveVel.Jerk := Parameters.Release.Jerk;
                Internal.MoveVel.Direction := Parameters.Release.Direction;
                Internal.MoveVel.BufferMode := Parameters.Release.BufferMode;

                Internal.State := slPOCKET_SYN_STATE_RESIZE_START;

            END_IF

        slPOCKET_SYN_STATE_RESIZE_START:

            IF NOT Enable THEN
                Internal.State := slPOCKET_SYN_STATE_RESET_FB;
            ELSIF Internal.StarCalcTarget.Error THEN
                Error := 1;
                ErrorID := Internal.StarCalcTarget.ErrorID;
                Internal.State := slPOCKET_SYN_STATE_RESET_FB;
            ELSIF Internal.ShReadInfo.Error THEN
                Error := 1;
                ErrorID := Internal.ShReadInfo.ErrorID;
                Internal.State := slPOCKET_SYN_STATE_RESET_FB;
            ELSIF Internal.Resize.Error THEN
                Error := 1;
                ErrorID := Internal.Resize.ErrorID;
                Internal.State := slPOCKET_SYN_STATE_RESET_FB;
            ELSIF Internal.Resize.Done THEN
                Internal.Resize.Execute := 0;
                IF Internal.StarCalcTarget.Valid THEN
                    Internal.CycPos.Enable := 1;
                    Internal.CycPos.CyclicPosition := Internal.StarCalcTarget.TrakPos;
                END_IF
                Internal.State := slPOCKET_SYN_STATE_SYNC;
            END_IF

        slPOCKET_SYN_STATE_SYNC:

            IF NOT Enable THEN
                Internal.State := slPOCKET_SYN_STATE_RESET_FB;
            ELSIF Internal.StarCalcTarget.Error THEN
                Error := 1;
                ErrorID := Internal.StarCalcTarget.ErrorID;
                Internal.State := slPOCKET_SYN_STATE_RESET_FB;
            ELSIF Internal.ShReadInfo.Error THEN
                Error := 1;
                ErrorID := Internal.ShReadInfo.ErrorID;
                Internal.State := slPOCKET_SYN_STATE_RESET_FB;
            ELSIF Internal.CycPos.Error THEN
                Error := 1;
                ErrorID := Internal.CycPos.ErrorID;
                Internal.State := slPOCKET_SYN_STATE_RESET_FB;
            //ELSIF Internal.CycPos.CommandAborted THEN
            //    Error := 1;
            //    ErrorID := slERR_SYNC_ABORTED;
            //    Internal.State := slPOCKET_SYN_STATE_RESET_FB;
            ELSIF Internal.StarCalcTarget.Valid THEN
                Internal.CycPos.Enable := 1;
                Internal.CycPos.CyclicPosition := Internal.StarCalcTarget.TrakPos;
                IF Internal.StarCalcTarget.TrakPos > Parameters.Release.Position THEN
                    Internal.MoveVel.Execute := 1;
                    Internal.State := slPOCKET_SYN_STATE_RELEASE;
                END_IF
            ELSE
                Internal.CycPos.Enable := 0;
                Internal.CycPos.CyclicPosition := 0;
            END_IF

        slPOCKET_SYN_STATE_RELEASE:

            IF NOT Enable THEN
                Internal.State := slPOCKET_SYN_STATE_RESET_FB;
            ELSIF Internal.StarCalcTarget.Error THEN
                Error := 1;
                ErrorID := Internal.StarCalcTarget.ErrorID;
                Internal.State := slPOCKET_SYN_STATE_RESET_FB;
            ELSIF Internal.ShReadInfo.Error THEN
                Error := 1;
                ErrorID := Internal.ShReadInfo.ErrorID;
                Internal.State := slPOCKET_SYN_STATE_RESET_FB;
            ELSIF Internal.CycPos.Error THEN
                Error := 1;
                ErrorID := Internal.CycPos.ErrorID;
                Internal.State := slPOCKET_SYN_STATE_RESET_FB;
            ELSIF Internal.MoveVel.Error THEN
                Error := 1;
                ErrorID := Internal.MoveVel.ErrorID;
                Internal.State := slPOCKET_SYN_STATE_RESET_FB;
            ELSIF Internal.MoveVel.Active THEN
                Internal.State := slPOCKET_SYN_STATE_WAIT_RESIZE;
            END_IF

        slPOCKET_SYN_STATE_WAIT_RESIZE:

            IF NOT Enable THEN
                Internal.State := slPOCKET_SYN_STATE_RESET_FB;
            ELSIF Internal.ShReadInfo.Error THEN
                Error := 1;
                ErrorID := Internal.ShReadInfo.ErrorID;
                Internal.State := slPOCKET_SYN_STATE_RESET_FB;
            ELSIF Internal.MoveVel.Error THEN
                Error := 1;
                ErrorID := Internal.MoveVel.ErrorID;
                Internal.State := slPOCKET_SYN_STATE_RESET_FB;
            ELSIF Internal.ShReadInfo.ShuttleInfo.CurrentValues.Position > Parameters.Release.ResizePosition THEN
                Internal.Resize.ResizeParameter := Parameters.ResizeEnd;
                Internal.Resize.Execute := 1;
                Internal.State := slPOCKET_SYN_STATE_RESIZE_END;
            END_IF

        slPOCKET_SYN_STATE_RESIZE_END:

            IF NOT Enable THEN
                Internal.State := slPOCKET_SYN_STATE_RESET_FB;
            ELSIF Internal.Resize.Error THEN
                Error := 1;
                ErrorID := Internal.Resize.ErrorID;
                Internal.State := slPOCKET_SYN_STATE_RESET_FB;
            ELSIF Internal.Resize.Done THEN
                Internal.CycPos.Enable := 0;
                Internal.ShReadInfo.Enable := 0;
                Internal.MoveVel.Execute := 0;
                Internal.Resize.Execute := 0;
                Done := 1;
                Internal.State := slPOCKET_SYN_STATE_DONE;
            END_IF

        slPOCKET_SYN_STATE_DONE:

            IF NOT Sync THEN
                Done := 0;
                Internal.State := slPOCKET_SYN_STATE_WAIT_SYNC;
            END_IF

        slPOCKET_SYN_STATE_RESET_FB:

            Sync := 0;
            Internal.StarCalcTarget.Enable := 0;
            Internal.ShReadInfo.Enable := 0;
            Internal.CycPos.Enable := 0;
            Internal.MoveVel.Execute := 0;
            Internal.Resize.Execute := 0;
            IF Error THEN
                Internal.State := slPOCKET_SYN_STATE_ERROR;
            ELSE
                Internal.State := slPOCKET_SYN_STATE_WAIT_NOT_BUSY;
            END_IF

        slPOCKET_SYN_STATE_WAIT_NOT_BUSY:

            IF NOT (Internal.ShReadInfo.Busy OR Internal.CycPos.Busy OR Internal.MoveVel.Busy OR Internal.Resize.Busy) THEN
                Busy := 0;
                Internal.State := slPOCKET_SYN_STATE_IDLE;
            END_IF

        slPOCKET_SYN_STATE_ERROR:

            IF NOT Enable THEN
                Error := 0;
                ErrorID := ERR_OK;
                Internal.State := slPOCKET_SYN_STATE_RESET_FB;
            END_IF

    END_CASE

    Internal.ShReadInfo();
    Internal.CycPos();
    Internal.MoveVel();
    Internal.Resize();

    InSync := Internal.CycPos.InCyclicPosition;
    Active := Enable AND Internal.StarCalcTarget.Valid AND NOT Error;

END_FUNCTION_BLOCK
